FUNCTION CheckDivInt : INT
VAR_INPUT
	divisor				: INT;
END_VAR
VAR
END_VAR

IF divisor = 0 THEN
	CheckIntZeroDiv_ErrCnt:= CheckIntZeroDiv_ErrCnt + 1;
	CheckDivInt := 1;
ELSE
	CheckDivInt := divisor;
END_IF

END_FUNCTION

(* stored: Version 1.1.0.1, ProductVersion 3.1.4024.9
   POU CheckDivInt: Id {c8f4c05e-212f-4904-97dd-e458963ed25b}, SpecialFunc CheckDivInt32 *)
